SPLINE
SPL {X  -159.452, Y  +378.767, Z    +0.000, E1   +11.887, E3 +156362.622}
SPL {X  -159.840, Y  +384.856, Z    +0.000, E1    +7.126, E3 +156381.593}
SPL {X  -159.991, Y  +390.336, Z    +0.000, E1    +2.803, E3 +156395.416}
SPL {X  -160.000, Y  +403.532, Z    +0.000, E1    -6.523, E3 +156413.137}
SPL {X  -160.000, Y  +409.023, Z    +0.000, E1   -10.003, E3 +156423.910}
SPL {X  -160.000, Y  +418.032, Z    +0.000, E1   -14.569, E3 +156448.770}
SPL {X  -160.000, Y  +420.561, Z    +0.000, E1   -14.816, E3 +156466.250}
SPL {X  -160.000, Y  +422.801, Z    +0.000, E1   -14.823, E3 +156484.198}
SPL {X  -160.000, Y  +425.518, Z    +0.000, E1   -14.845, E3 +156505.973}
SPL {X  -160.000, Y  +428.688, Z    +0.000, E1   -14.854, E3 +156531.381}
SPL {X  -160.000, Y  +431.971, Z    +0.000, E1   -14.849, E3 +156557.850}
SPL {X  -160.000, Y  +435.345, Z    +0.000, E1   -14.857, E3 +156584.900}
SPL {X  -160.000, Y  +438.732, Z    +0.000, E1   -14.858, E3 +156612.048}
SPL {X  -160.000, Y  +441.925, Z    +0.000, E1   -14.848, E3 +156637.718}
SPL {X  -160.000, Y  +444.299, Z    +0.000, E1   -14.809, E3 +156656.903}
SPL {X  -160.000, Y  +446.229, Z    +0.000, E1   -14.820, E3 +156672.322}
SPL {X  -160.000, Y  +448.987, Z    +0.000, E1   -14.868, E3 +156694.259}
SPL {X  -160.000, Y  +452.351, Z    +0.000, E1   -14.871, E3 +156721.235}
SPL {X  -160.000, Y  +455.709, Z    +0.000, E1   -14.880, E3 +156748.049}
SPL {X  -160.000, Y  +458.189, Z    +0.000, E1   -14.832, E3 +156768.051}
SPL {X  -160.000, Y  +459.885, Z    +0.000, E1   -14.825, E3 +156781.721}
SPL {X  -160.000, Y  +462.438, Z    +0.000, E1   -14.868, E3 +156802.131}
SPL {X  -160.000, Y  +465.575, Z    +0.000, E1   -14.849, E3 +156827.439}
SPL {X  -160.000, Y  +468.581, Z    +0.000, E1   -14.841, E3 +156851.672}
SPL {X  -160.000, Y  +471.795, Z    +0.000, E1   -14.854, E3 +156877.459}
SPL {X  -160.000, Y  +475.138, Z    +0.000, E1   -14.853, E3 +156904.310}
SPL {X  -160.000, Y  +477.981, Z    +0.000, E1   -14.823, E3 +156927.230}
SPL {X  -160.000, Y  +480.658, Z    +0.000, E1   -14.835, E3 +156948.706}
SPL {X  -160.000, Y  +483.534, Z    +0.000, E1   -14.838, E3 +156971.801}
SPL {X  -160.000, Y  +486.226, Z    +0.000, E1   -14.823, E3 +156993.466}
SPL {X  -160.000, Y  +488.751, Z    +0.000, E1   -14.827, E3 +157013.738}
SPL {X  -160.000, Y  +491.612, Z    +0.000, E1   -14.844, E3 +157036.661}
SPL {X  -160.000, Y  +494.417, Z    +0.000, E1   -14.827, E3 +157059.252}
SPL {X  -160.000, Y  +496.961, Z    +0.000, E1   -14.824, E3 +157079.696}
SPL {X  -160.000, Y  +499.610, Z    +0.000, E1   -14.830, E3 +157100.968}
SPL {X  -160.000, Y  +502.268, Z    +0.000, E1   -14.832, E3 +157122.238}
SPL {X  -160.000, Y  +505.041, Z    +0.000, E1   -14.849, E3 +157144.400}
SPL {X  -160.000, Y  +507.743, Z    +0.000, E1   -14.842, E3 +157166.024}
SPL {X  -160.000, Y  +510.437, Z    +0.000, E1   -14.860, E3 +157187.538}
SPL {X  -160.000, Y  +513.179, Z    +0.000, E1   -14.849, E3 +157209.585}
SPL {X  -160.000, Y  +515.613, Z    +0.000, E1   -14.829, E3 +157229.256}
SPL {X  -160.000, Y  +518.188, Z    +0.000, E1   -14.845, E3 +157249.885}
SPL {X  -160.000, Y  +520.790, Z    +0.000, E1   -14.839, E3 +157270.714}
SPL {X  -160.000, Y  +523.469, Z    +0.000, E1   -14.855, E3 +157292.162}
SPL {X  -160.000, Y  +526.403, Z    +0.000, E1   -14.858, E3 +157315.698}
SPL {X  -160.000, Y  +529.266, Z    +0.000, E1   -14.848, E3 +157338.706}
SPL {X  -160.000, Y  +531.688, Z    +0.000, E1   -14.826, E3 +157358.255}
SPL {X  -160.000, Y  +534.214, Z    +0.000, E1   -14.841, E3 +157378.518}
SPL {X  -160.000, Y  +537.002, Z    +0.000, E1   -14.839, E3 +157400.937}
SPL {X  -160.000, Y  +539.729, Z    +0.000, E1   -14.840, E3 +157422.748}
SPL {X  -160.000, Y  +542.408, Z    +0.000, E1   -14.839, E3 +157444.301}
SPL {X  -160.000, Y  +545.014, Z    +0.000, E1   -14.831, E3 +157465.246}
SPL {X  -160.000, Y  +547.659, Z    +0.000, E1   -14.839, E3 +157486.461}
SPL {X  -160.000, Y  +550.215, Z    +0.000, E1   -14.827, E3 +157507.026}
SPL {X  -160.000, Y  +552.762, Z    +0.000, E1   -14.836, E3 +157527.444}
SPL {X  -160.000, Y  +555.331, Z    +0.000, E1   -14.837, E3 +157547.985}
SPL {X  -160.000, Y  +558.235, Z    +0.000, E1   -14.869, E3 +157571.149}
SPL {X  -160.000, Y  +561.088, Z    +0.000, E1   -14.848, E3 +157594.067}
SPL {X  -160.000, Y  +563.693, Z    +0.000, E1   -14.852, E3 +157614.928}
SPL {X  -160.000, Y  +566.560, Z    +0.000, E1   -14.865, E3 +157637.905}
SPL {X  -160.000, Y  +569.305, Z    +0.000, E1   -14.848, E3 +157659.934}
SPL {X  -160.000, Y  +571.769, Z    +0.000, E1   -14.852, E3 +157679.680}
SPL {X  -160.000, Y  +574.366, Z    +0.000, E1   -14.855, E3 +157700.467}
SPL {X  -160.000, Y  +577.037, Z    +0.000, E1   -14.859, E3 +157721.866}
SPL {X  -160.000, Y  +579.855, Z    +0.000, E1   -14.869, E3 +157744.393}
SPL {X  -160.000, Y  +582.456, Z    +0.000, E1   -14.854, E3 +157765.253}
SPL {X  -160.000, Y  +585.083, Z    +0.000, E1   -14.866, E3 +157786.303}
SPL {X  -160.000, Y  +587.675, Z    +0.000, E1   -14.853, E3 +157807.094}
SPL {X  -160.000, Y  +590.216, Z    +0.000, E1   -14.864, E3 +157827.413}
SPL {X  -160.000, Y  +592.848, Z    +0.000, E1   -14.865, E3 +157848.464}
SPL {X  -160.000, Y  +595.342, Z    +0.000, E1   -14.848, E3 +157868.642}
SPL {X  -160.000, Y  +597.995, Z    +0.000, E1   -14.848, E3 +157889.982}
SPL {X  -160.000, Y  +600.731, Z    +0.000, E1   -14.846, E3 +157911.933}
SPL {X  -160.000, Y  +603.404, Z    +0.000, E1   -14.846, E3 +157933.369}
SPL {X  -160.000, Y  +605.923, Z    +0.000, E1   -14.838, E3 +157953.610}
SPL {X  -160.000, Y  +608.492, Z    +0.000, E1   -14.846, E3 +157974.214}
SPL {X  -160.000, Y  +611.345, Z    +0.000, E1   -14.856, E3 +157997.072}
SPL {X  -160.000, Y  +614.087, Z    +0.000, E1   -14.839, E3 +158019.131}
SPL {X  -160.000, Y  +616.566, Z    +0.000, E1   -14.839, E3 +158039.025}
SPL {X  -160.000, Y  +619.350, Z    +0.000, E1   -14.855, E3 +158061.313}
SPL {X  -160.000, Y  +622.198, Z    +0.000, E1   -14.846, E3 +158084.197}
SPL {X  -160.000, Y  +624.642, Z    +0.000, E1   -14.829, E3 +158103.870}
SPL {X  -160.000, Y  +627.119, Z    +0.000, E1   -14.843, E3 +158123.710}
SPL {X  -160.000, Y  +629.682, Z    +0.000, E1   -14.838, E3 +158144.279}
SPL {X  -160.000, Y  +632.223, Z    +0.000, E1   -14.841, E3 +158164.670}
SPL {X  -160.000, Y  +634.941, Z    +0.000, E1   -14.846, E3 +158186.468}
SPL {X  -160.000, Y  +637.723, Z    +0.000, E1   -14.844, E3 +158208.812}
SPL {X  -160.000, Y  +640.315, Z    +0.000, E1   -14.836, E3 +158229.610}
SPL {X  -160.000, Y  +643.085, Z    +0.000, E1   -14.865, E3 +158251.661}
SPL {X  -160.000, Y  +645.845, Z    +0.000, E1   -14.848, E3 +158273.849}
SPL {X  -160.000, Y  +648.229, Z    +0.000, E1   -14.834, E3 +158293.059}
SPL {X  -160.000, Y  +650.656, Z    +0.000, E1   -14.835, E3 +158312.615}
SPL {X  -160.000, Y  +653.134, Z    +0.000, E1   -14.827, E3 +158332.542}
SPL {X  -160.000, Y  +655.670, Z    +0.000, E1   -14.841, E3 +158352.836}
SPL {X  -160.000, Y  +658.349, Z    +0.000, E1   -14.842, E3 +158374.312}
SPL {X  -160.000, Y  +660.936, Z    +0.000, E1   -14.838, E3 +158395.064}
SPL {X  -160.000, Y  +663.567, Z    +0.000, E1   -14.845, E3 +158416.194}
SPL {X  -160.000, Y  +666.216, Z    +0.000, E1   -14.832, E3 +158437.511}
SPL {X  -159.997, Y  +668.731, Z    +0.000, E1   -14.834, E3 +158457.703}
SPL {X  -159.962, Y  +671.176, Z    +0.000, E1   -14.822, E3 +158477.414}
SPL {X  -159.895, Y  +673.507, Z    +0.000, E1   -14.821, E3 +158496.145}
SPL {X  -159.785, Y  +675.985, Z    +0.000, E1   -14.818, E3 +158516.147}
SPL {X  -159.627, Y  +678.622, Z    +0.000, E1   -14.804, E3 +158537.500}
SPL {X  -159.438, Y  +681.094, Z    +0.000, E1   -14.770, E3 +158557.671}
SPL {X  -159.262, Y  +683.054, Z    +0.000, E1   -14.719, E3 +158573.899}
ENDSPLINE

SPLINE
SPL {X  -159.661, Y  +678.114, Z    +0.000, E1    -9.575, E3 +158603.491}
SPL {X  -159.942, Y  +672.020, Z    +0.000, E1    -4.692, E3 +158622.118}
SPL {X  -160.000, Y  +664.971, Z    +0.000, E1    +0.516, E3 +158641.668}
SPL {X  -160.000, Y  +660.032, Z    +0.000, E1    +3.995, E3 +158653.611}
SPL {X  -160.000, Y  +652.280, Z    +0.000, E1    +8.913, E3 +158672.126}
SPL {X  -160.000, Y  +644.147, Z    +0.000, E1   +13.158, E3 +158695.677}
SPL {X  -160.000, Y  +641.594, Z    +0.000, E1   +13.488, E3 +158714.118}
SPL {X  -160.000, Y  +639.799, Z    +0.000, E1   +13.486, E3 +158730.028}
SPL {X  -160.000, Y  +637.896, Z    +0.000, E1   +13.493, E3 +158746.843}
SPL {X  -160.000, Y  +635.832, Z    +0.000, E1   +13.499, E3 +158765.102}
SPL {X  -160.000, Y  +633.839, Z    +0.000, E1   +13.489, E3 +158782.790}
SPL {X  -160.000, Y  +631.625, Z    +0.000, E1   +13.508, E3 +158802.331}
SPL {X  -160.000, Y  +629.417, Z    +0.000, E1   +13.491, E3 +158821.943}
SPL {X  -160.000, Y  +627.180, Z    +0.000, E1   +13.508, E3 +158841.697}
SPL {X  -160.000, Y  +624.970, Z    +0.000, E1   +13.490, E3 +158861.347}
SPL {X  -160.000, Y  +623.020, Z    +0.000, E1   +13.491, E3 +158878.576}
SPL {X  -160.000, Y  +620.888, Z    +0.000, E1   +13.501, E3 +158897.439}
SPL {X  -160.000, Y  +618.790, Z    +0.000, E1   +13.488, E3 +158916.061}
SPL {X  -160.000, Y  +616.631, Z    +0.000, E1   +13.504, E3 +158935.115}
SPL {X  -160.000, Y  +614.230, Z    +0.000, E1   +13.510, E3 +158956.311}
SPL {X  -160.000, Y  +612.132, Z    +0.000, E1   +13.485, E3 +158975.027}
SPL {X  -160.000, Y  +610.405, Z    +0.000, E1   +13.477, E3 +158990.400}
SPL {X  -160.000, Y  +608.437, Z    +0.000, E1   +13.502, E3 +159007.656}
SPL {X  -160.000, Y  +606.281, Z    +0.000, E1   +13.502, E3 +159026.673}
SPL {X  -160.000, Y  +604.124, Z    +0.000, E1   +13.513, E3 +159045.729}
SPL {X  -160.000, Y  +601.878, Z    +0.000, E1   +13.505, E3 +159065.626}
SPL {X  -160.000, Y  +599.648, Z    +0.000, E1   +13.506, E3 +159085.403}
SPL {X  -160.000, Y  +597.673, Z    +0.000, E1   +13.479, E3 +159103.076}
SPL {X  -160.000, Y  +595.601, Z    +0.000, E1   +13.499, E3 +159121.359}
SPL {X  -160.000, Y  +593.187, Z    +0.000, E1   +13.500, E3 +159142.739}
SPL {X  -160.000, Y  +591.079, Z    +0.000, E1   +13.483, E3 +159161.466}
SPL {X  -160.000, Y  +589.151, Z    +0.000, E1   +13.489, E3 +159178.517}
SPL {X  -160.000, Y  +586.908, Z    +0.000, E1   +13.501, E3 +159198.362}
SPL {X  -160.000, Y  +584.660, Z    +0.000, E1   +13.490, E3 +159218.304}
SPL {X  -160.000, Y  +582.409, Z    +0.000, E1   +13.499, E3 +159238.222}
SPL {X  -160.000, Y  +580.150, Z    +0.000, E1   +13.490, E3 +159258.268}
SPL {X  -160.000, Y  +577.953, Z    +0.000, E1   +13.493, E3 +159277.727}
SPL {X  -160.000, Y  +575.630, Z    +0.000, E1   +13.502, E3 +159298.211}
SPL {X  -160.000, Y  +573.418, Z    +0.000, E1   +13.502, E3 +159317.719}
SPL {X  -160.000, Y  +571.226, Z    +0.000, E1   +13.520, E3 +159336.927}
SPL {X  -160.000, Y  +569.166, Z    +0.000, E1   +13.512, E3 +159355.118}
SPL {X  -160.000, Y  +567.275, Z    +0.000, E1   +13.517, E3 +159371.785}
SPL {X  -160.000, Y  +565.259, Z    +0.000, E1   +13.523, E3 +159389.574}
SPL {X  -160.000, Y  +563.305, Z    +0.000, E1   +13.512, E3 +159406.913}
SPL {X  -160.000, Y  +561.240, Z    +0.000, E1   +13.521, E3 +159425.174}
SPL {X  -160.000, Y  +558.881, Z    +0.000, E1   +13.524, E3 +159446.016}
SPL {X  -160.000, Y  +556.697, Z    +0.000, E1   +13.510, E3 +159465.402}
SPL {X  -160.000, Y  +554.624, Z    +0.000, E1   +13.512, E3 +159483.733}
SPL {X  -160.000, Y  +552.465, Z    +0.000, E1   +13.514, E3 +159502.818}
SPL {X  -160.000, Y  +550.315, Z    +0.000, E1   +13.514, E3 +159521.811}
SPL {X  -160.000, Y  +548.056, Z    +0.000, E1   +13.519, E3 +159541.812}
SPL {X  -160.000, Y  +545.826, Z    +0.000, E1   +13.501, E3 +159561.690}
SPL {X  -160.000, Y  +543.677, Z    +0.000, E1   +13.502, E3 +159580.748}
SPL {X  -160.000, Y  +541.664, Z    +0.000, E1   +13.489, E3 +159598.633}
SPL {X  -160.000, Y  +539.659, Z    +0.000, E1   +13.494, E3 +159616.393}
SPL {X  -160.000, Y  +537.370, Z    +0.000, E1   +13.501, E3 +159636.632}
SPL {X  -160.000, Y  +535.056, Z    +0.000, E1   +13.506, E3 +159657.028}
SPL {X  -160.000, Y  +532.975, Z    +0.000, E1   +13.494, E3 +159675.515}
SPL {X  -160.000, Y  +530.925, Z    +0.000, E1   +13.499, E3 +159693.676}
SPL {X  -160.000, Y  +528.768, Z    +0.000, E1   +13.498, E3 +159712.778}
SPL {X  -160.000, Y  +526.547, Z    +0.000, E1   +13.499, E3 +159732.446}
SPL {X  -160.000, Y  +523.964, Z    +0.000, E1   +13.742, E3 +159751.951}
SPL {X  -160.000, Y  +513.971, Z    +0.000, E1   +18.644, E3 +159770.863}
SPL {X  -160.000, Y  +513.562, Z    +0.000, E1   +16.972, E3 +159790.740}
SPL {X  -160.000, Y  +513.358, Z    +0.000, E1   +15.267, E3 +159811.012}
SPL {X  -160.000, Y  +512.244, Z    +0.000, E1   +14.473, E3 +159829.468}
SPL {X  -160.000, Y  +509.675, Z    +0.000, E1   +14.481, E3 +159850.611}
SPL {X  -160.000, Y  +507.162, Z    +0.000, E1   +14.470, E3 +159871.351}
SPL {X  -160.000, Y  +504.735, Z    +0.000, E1   +14.473, E3 +159891.323}
SPL {X  -160.000, Y  +502.261, Z    +0.000, E1   +14.476, E3 +159911.659}
SPL {X  -160.000, Y  +499.798, Z    +0.000, E1   +14.482, E3 +159931.861}
SPL {X  -160.000, Y  +497.435, Z    +0.000, E1   +14.476, E3 +159951.338}
SPL {X  -160.000, Y  +495.089, Z    +0.000, E1   +14.475, E3 +159970.705}
SPL {X  -160.000, Y  +492.764, Z    +0.000, E1   +14.469, E3 +159989.876}
SPL {X  -160.000, Y  +490.292, Z    +0.000, E1   +14.476, E3 +160010.277}
SPL {X  -160.000, Y  +487.641, Z    +0.000, E1   +14.470, E3 +160032.173}
SPL {X  -160.000, Y  +485.054, Z    +0.000, E1   +14.460, E3 +160053.616}
SPL {X  -160.000, Y  +482.421, Z    +0.000, E1   +14.461, E3 +160075.334}
SPL {X  -160.000, Y  +480.000, Z    +0.000, E1   +14.451, E3 +160095.298}
SPL {X  -160.000, Y  +477.551, Z    +0.000, E1   +14.466, E3 +160115.427}
SPL {X  -160.000, Y  +475.253, Z    +0.000, E1   +14.450, E3 +160134.401}
SPL {X  -160.000, Y  +473.070, Z    +0.000, E1   +14.454, E3 +160152.422}
SPL {X  -160.000, Y  +470.603, Z    +0.000, E1   +14.464, E3 +160172.722}
SPL {X  -160.000, Y  +468.243, Z    +0.000, E1   +14.458, E3 +160192.121}
SPL {X  -160.000, Y  +465.791, Z    +0.000, E1   +14.475, E3 +160212.265}
SPL {X  -160.000, Y  +463.103, Z    +0.000, E1   +14.474, E3 +160234.414}
SPL {X  -160.000, Y  +460.743, Z    +0.000, E1   +14.465, E3 +160253.822}
SPL {X  -160.000, Y  +458.292, Z    +0.000, E1   +14.492, E3 +160273.822}
SPL {X  -160.000, Y  +455.874, Z    +0.000, E1   +14.484, E3 +160293.679}
SPL {X  -160.000, Y  +453.555, Z    +0.000, E1   +14.488, E3 +160312.759}
SPL {X  -160.000, Y  +451.093, Z    +0.000, E1   +14.485, E3 +160333.071}
SPL {X  -160.000, Y  +448.700, Z    +0.000, E1   +14.483, E3 +160352.760}
SPL {X  -160.000, Y  +446.277, Z    +0.000, E1   +14.485, E3 +160372.684}
SPL {X  -160.000, Y  +443.879, Z    +0.000, E1   +14.485, E3 +160392.422}
SPL {X  -160.000, Y  +441.447, Z    +0.000, E1   +14.485, E3 +160412.429}
SPL {X  -160.000, Y  +439.006, Z    +0.000, E1   +14.488, E3 +160432.512}
SPL {X  -160.000, Y  +436.311, Z    +0.000, E1   +14.498, E3 +160454.671}
SPL {X  -160.000, Y  +433.559, Z    +0.000, E1   +14.491, E3 +160477.341}
SPL {X  -160.000, Y  +431.162, Z    +0.000, E1   +14.479, E3 +160497.092}
SPL {X  -160.000, Y  +429.152, Z    +0.000, E1   +14.469, E3 +160513.673}
SPL {X  -160.000, Y  +426.863, Z    +0.000, E1   +14.490, E3 +160532.452}
SPL {X  -160.000, Y  +424.653, Z    +0.000, E1   +14.467, E3 +160550.712}
SPL {X  -160.000, Y  +422.337, Z    +0.000, E1   +14.492, E3 +160569.696}
SPL {X  -160.000, Y  +419.639, Z    +0.000, E1   +14.504, E3 +160591.736}
SPL {X  -160.000, Y  +417.127, Z    +0.000, E1   +14.501, E3 +160612.327}
SPL {X  -160.000, Y  +414.849, Z    +0.000, E1   +14.496, E3 +160631.061}
SPL {X  -160.000, Y  +412.396, Z    +0.000, E1   +14.505, E3 +160651.250}
SPL {X  -160.000, Y  +409.815, Z    +0.000, E1   +14.498, E3 +160672.504}
SPL {X  -160.000, Y  +407.614, Z    +0.000, E1   +14.484, E3 +160690.629}
SPL {X  -160.000, Y  +405.406, Z    +0.000, E1   +14.501, E3 +160708.692}
SPL {X  -160.000, Y  +402.958, Z    +0.000, E1   +14.500, E3 +160728.862}
SPL {X  -160.000, Y  +400.690, Z    +0.000, E1   +14.484, E3 +160747.574}
SPL {X  -160.000, Y  +398.391, Z    +0.000, E1   +14.502, E3 +160766.400}
SPL {X  -160.000, Y  +395.999, Z    +0.000, E1   +14.484, E3 +160786.190}
SPL {X  -160.000, Y  +393.685, Z    +0.000, E1   +14.486, E3 +160805.262}
SPL {X  -159.999, Y  +391.313, Z    +0.000, E1   +14.479, E3 +160824.844}
SPL {X  -159.970, Y  +388.900, Z    +0.000, E1   +14.480, E3 +160844.729}
SPL {X  -159.903, Y  +386.417, Z    +0.000, E1   +14.475, E3 +160865.234}
SPL {X  -159.796, Y  +383.921, Z    +0.000, E1   +14.466, E3 +160885.889}
SPL {X  -159.651, Y  +381.443, Z    +0.000, E1   +14.453, E3 +160906.437}
SPL {X  -159.474, Y  +379.042, Z    +0.000, E1   +14.434, E3 +160926.401}
SPL {X  -159.316, Y  +377.219, Z    +0.000, E1   +14.400, E3 +160941.629}
ENDSPLINE

SPLINE
SPL {X  -159.452, Y  +378.767, Z    +0.000, E1   +11.887, E3 +160962.619}
SPL {X  -159.840, Y  +384.856, Z    +0.000, E1    +7.126, E3 +160981.590}
SPL {X  -159.991, Y  +390.336, Z    +0.000, E1    +2.803, E3 +160995.413}
SPL {X  -160.000, Y  +403.532, Z    +0.000, E1    -6.523, E3 +161013.134}
SPL {X  -160.000, Y  +409.023, Z    +0.000, E1   -10.003, E3 +161023.907}
SPL {X  -160.000, Y  +418.032, Z    +0.000, E1   -14.569, E3 +161048.766}
SPL {X  -160.000, Y  +420.561, Z    +0.000, E1   -14.816, E3 +161066.246}
SPL {X  -160.000, Y  +422.801, Z    +0.000, E1   -14.823, E3 +161084.195}
SPL {X  -160.000, Y  +425.518, Z    +0.000, E1   -14.845, E3 +161105.970}
SPL {X  -160.000, Y  +428.688, Z    +0.000, E1   -14.854, E3 +161131.378}
SPL {X  -160.000, Y  +431.971, Z    +0.000, E1   -14.849, E3 +161157.846}
SPL {X  -160.000, Y  +435.345, Z    +0.000, E1   -14.857, E3 +161184.897}
SPL {X  -160.000, Y  +438.732, Z    +0.000, E1   -14.858, E3 +161212.045}
SPL {X  -160.000, Y  +441.925, Z    +0.000, E1   -14.848, E3 +161237.715}
SPL {X  -160.000, Y  +444.299, Z    +0.000, E1   -14.809, E3 +161256.900}
SPL {X  -160.000, Y  +446.229, Z    +0.000, E1   -14.820, E3 +161272.319}
SPL {X  -160.000, Y  +448.987, Z    +0.000, E1   -14.868, E3 +161294.256}
SPL {X  -160.000, Y  +452.351, Z    +0.000, E1   -14.871, E3 +161321.232}
SPL {X  -160.000, Y  +455.709, Z    +0.000, E1   -14.880, E3 +161348.046}
SPL {X  -160.000, Y  +458.189, Z    +0.000, E1   -14.832, E3 +161368.047}
SPL {X  -160.000, Y  +459.885, Z    +0.000, E1   -14.825, E3 +161381.718}
SPL {X  -160.000, Y  +462.438, Z    +0.000, E1   -14.868, E3 +161402.128}
SPL {X  -160.000, Y  +465.575, Z    +0.000, E1   -14.849, E3 +161427.436}
SPL {X  -160.000, Y  +468.581, Z    +0.000, E1   -14.841, E3 +161451.669}
SPL {X  -160.000, Y  +471.795, Z    +0.000, E1   -14.854, E3 +161477.456}
SPL {X  -160.000, Y  +475.138, Z    +0.000, E1   -14.853, E3 +161504.306}
SPL {X  -160.000, Y  +477.981, Z    +0.000, E1   -14.823, E3 +161527.227}
SPL {X  -160.000, Y  +480.658, Z    +0.000, E1   -14.835, E3 +161548.703}
SPL {X  -160.000, Y  +483.534, Z    +0.000, E1   -14.838, E3 +161571.798}
SPL {X  -160.000, Y  +486.226, Z    +0.000, E1   -14.823, E3 +161593.463}
SPL {X  -160.000, Y  +488.751, Z    +0.000, E1   -14.827, E3 +161613.735}
SPL {X  -160.000, Y  +491.612, Z    +0.000, E1   -14.844, E3 +161636.658}
SPL {X  -160.000, Y  +494.417, Z    +0.000, E1   -14.827, E3 +161659.249}
SPL {X  -160.000, Y  +496.961, Z    +0.000, E1   -14.824, E3 +161679.692}
SPL {X  -160.000, Y  +499.610, Z    +0.000, E1   -14.830, E3 +161700.965}
SPL {X  -160.000, Y  +502.268, Z    +0.000, E1   -14.832, E3 +161722.234}
SPL {X  -160.000, Y  +505.041, Z    +0.000, E1   -14.849, E3 +161744.397}
SPL {X  -160.000, Y  +507.743, Z    +0.000, E1   -14.842, E3 +161766.021}
SPL {X  -160.000, Y  +510.437, Z    +0.000, E1   -14.860, E3 +161787.535}
SPL {X  -160.000, Y  +513.179, Z    +0.000, E1   -14.849, E3 +161809.582}
SPL {X  -160.000, Y  +515.613, Z    +0.000, E1   -14.829, E3 +161829.252}
SPL {X  -160.000, Y  +518.188, Z    +0.000, E1   -14.845, E3 +161849.882}
SPL {X  -160.000, Y  +520.790, Z    +0.000, E1   -14.839, E3 +161870.711}
SPL {X  -160.000, Y  +523.469, Z    +0.000, E1   -14.855, E3 +161892.159}
SPL {X  -160.000, Y  +526.403, Z    +0.000, E1   -14.858, E3 +161915.695}
SPL {X  -160.000, Y  +529.266, Z    +0.000, E1   -14.848, E3 +161938.702}
SPL {X  -160.000, Y  +531.688, Z    +0.000, E1   -14.826, E3 +161958.252}
SPL {X  -160.000, Y  +534.214, Z    +0.000, E1   -14.841, E3 +161978.515}
SPL {X  -160.000, Y  +537.002, Z    +0.000, E1   -14.839, E3 +162000.933}
SPL {X  -160.000, Y  +539.729, Z    +0.000, E1   -14.840, E3 +162022.745}
SPL {X  -160.000, Y  +542.408, Z    +0.000, E1   -14.839, E3 +162044.298}
SPL {X  -160.000, Y  +545.014, Z    +0.000, E1   -14.831, E3 +162065.243}
SPL {X  -160.000, Y  +547.659, Z    +0.000, E1   -14.839, E3 +162086.458}
SPL {X  -160.000, Y  +550.215, Z    +0.000, E1   -14.827, E3 +162107.023}
SPL {X  -160.000, Y  +552.762, Z    +0.000, E1   -14.836, E3 +162127.441}
SPL {X  -160.000, Y  +555.331, Z    +0.000, E1   -14.837, E3 +162147.982}
SPL {X  -160.000, Y  +558.235, Z    +0.000, E1   -14.869, E3 +162171.145}
SPL {X  -160.000, Y  +561.088, Z    +0.000, E1   -14.848, E3 +162194.064}
SPL {X  -160.000, Y  +563.693, Z    +0.000, E1   -14.852, E3 +162214.924}
SPL {X  -160.000, Y  +566.560, Z    +0.000, E1   -14.865, E3 +162237.902}
SPL {X  -160.000, Y  +569.305, Z    +0.000, E1   -14.848, E3 +162259.931}
SPL {X  -160.000, Y  +571.769, Z    +0.000, E1   -14.852, E3 +162279.676}
SPL {X  -160.000, Y  +574.366, Z    +0.000, E1   -14.855, E3 +162300.463}
SPL {X  -160.000, Y  +577.037, Z    +0.000, E1   -14.859, E3 +162321.863}
SPL {X  -160.000, Y  +579.855, Z    +0.000, E1   -14.869, E3 +162344.390}
SPL {X  -160.000, Y  +582.456, Z    +0.000, E1   -14.854, E3 +162365.250}
SPL {X  -160.000, Y  +585.083, Z    +0.000, E1   -14.866, E3 +162386.300}
SPL {X  -160.000, Y  +587.675, Z    +0.000, E1   -14.853, E3 +162407.091}
SPL {X  -160.000, Y  +590.216, Z    +0.000, E1   -14.864, E3 +162427.410}
SPL {X  -160.000, Y  +592.848, Z    +0.000, E1   -14.865, E3 +162448.461}
SPL {X  -160.000, Y  +595.342, Z    +0.000, E1   -14.848, E3 +162468.639}
SPL {X  -160.000, Y  +597.995, Z    +0.000, E1   -14.848, E3 +162489.979}
SPL {X  -160.000, Y  +600.731, Z    +0.000, E1   -14.846, E3 +162511.930}
SPL {X  -160.000, Y  +603.404, Z    +0.000, E1   -14.846, E3 +162533.366}
SPL {X  -160.000, Y  +605.923, Z    +0.000, E1   -14.838, E3 +162553.607}
SPL {X  -160.000, Y  +608.492, Z    +0.000, E1   -14.846, E3 +162574.210}
SPL {X  -160.000, Y  +611.345, Z    +0.000, E1   -14.856, E3 +162597.069}
SPL {X  -160.000, Y  +614.087, Z    +0.000, E1   -14.839, E3 +162619.128}
SPL {X  -160.000, Y  +616.566, Z    +0.000, E1   -14.839, E3 +162639.022}
SPL {X  -160.000, Y  +619.350, Z    +0.000, E1   -14.855, E3 +162661.310}
SPL {X  -160.000, Y  +622.198, Z    +0.000, E1   -14.846, E3 +162684.194}
SPL {X  -160.000, Y  +624.642, Z    +0.000, E1   -14.829, E3 +162703.867}
SPL {X  -160.000, Y  +627.119, Z    +0.000, E1   -14.843, E3 +162723.707}
SPL {X  -160.000, Y  +629.682, Z    +0.000, E1   -14.838, E3 +162744.276}
SPL {X  -160.000, Y  +632.223, Z    +0.000, E1   -14.841, E3 +162764.667}
SPL {X  -160.000, Y  +634.941, Z    +0.000, E1   -14.846, E3 +162786.465}
SPL {X  -160.000, Y  +637.723, Z    +0.000, E1   -14.844, E3 +162808.809}
SPL {X  -160.000, Y  +640.315, Z    +0.000, E1   -14.836, E3 +162829.606}
SPL {X  -160.000, Y  +643.085, Z    +0.000, E1   -14.865, E3 +162851.658}
SPL {X  -160.000, Y  +645.845, Z    +0.000, E1   -14.848, E3 +162873.846}
SPL {X  -160.000, Y  +648.229, Z    +0.000, E1   -14.834, E3 +162893.056}
SPL {X  -160.000, Y  +650.656, Z    +0.000, E1   -14.835, E3 +162912.612}
SPL {X  -160.000, Y  +653.134, Z    +0.000, E1   -14.827, E3 +162932.539}
SPL {X  -160.000, Y  +655.670, Z    +0.000, E1   -14.841, E3 +162952.833}
SPL {X  -160.000, Y  +658.349, Z    +0.000, E1   -14.842, E3 +162974.309}
SPL {X  -160.000, Y  +660.936, Z    +0.000, E1   -14.838, E3 +162995.061}
SPL {X  -160.000, Y  +663.567, Z    +0.000, E1   -14.845, E3 +163016.191}
SPL {X  -160.000, Y  +666.216, Z    +0.000, E1   -14.832, E3 +163037.508}
SPL {X  -159.997, Y  +668.731, Z    +0.000, E1   -14.834, E3 +163057.700}
SPL {X  -159.962, Y  +671.176, Z    +0.000, E1   -14.822, E3 +163077.411}
SPL {X  -159.895, Y  +673.507, Z    +0.000, E1   -14.821, E3 +163096.142}
SPL {X  -159.785, Y  +675.985, Z    +0.000, E1   -14.818, E3 +163116.144}
SPL {X  -159.627, Y  +678.622, Z    +0.000, E1   -14.804, E3 +163137.496}
SPL {X  -159.438, Y  +681.094, Z    +0.000, E1   -14.770, E3 +163157.668}
SPL {X  -159.262, Y  +683.054, Z    +0.000, E1   -14.719, E3 +163173.896}
ENDSPLINE

SPLINE
SPL {X  -159.661, Y  +678.114, Z    +0.000, E1    -9.575, E3 +163203.488}
SPL {X  -159.942, Y  +672.020, Z    +0.000, E1    -4.692, E3 +163222.115}
SPL {X  -160.000, Y  +664.971, Z    +0.000, E1    +0.516, E3 +163241.665}
SPL {X  -160.000, Y  +660.032, Z    +0.000, E1    +3.995, E3 +163253.608}
SPL {X  -160.000, Y  +652.280, Z    +0.000, E1    +8.913, E3 +163272.123}
SPL {X  -160.000, Y  +644.147, Z    +0.000, E1   +13.158, E3 +163295.674}
SPL {X  -160.000, Y  +641.594, Z    +0.000, E1   +13.488, E3 +163314.115}
SPL {X  -160.000, Y  +639.799, Z    +0.000, E1   +13.486, E3 +163330.025}
SPL {X  -160.000, Y  +637.896, Z    +0.000, E1   +13.493, E3 +163346.840}
SPL {X  -160.000, Y  +635.832, Z    +0.000, E1   +13.499, E3 +163365.098}
SPL {X  -160.000, Y  +633.839, Z    +0.000, E1   +13.489, E3 +163382.787}
SPL {X  -160.000, Y  +631.625, Z    +0.000, E1   +13.508, E3 +163402.328}
SPL {X  -160.000, Y  +629.417, Z    +0.000, E1   +13.491, E3 +163421.939}
SPL {X  -160.000, Y  +627.180, Z    +0.000, E1   +13.508, E3 +163441.693}
SPL {X  -160.000, Y  +624.970, Z    +0.000, E1   +13.490, E3 +163461.343}
SPL {X  -160.000, Y  +623.020, Z    +0.000, E1   +13.491, E3 +163478.573}
SPL {X  -160.000, Y  +620.888, Z    +0.000, E1   +13.501, E3 +163497.436}
SPL {X  -160.000, Y  +618.790, Z    +0.000, E1   +13.488, E3 +163516.058}
SPL {X  -160.000, Y  +616.631, Z    +0.000, E1   +13.504, E3 +163535.112}
SPL {X  -160.000, Y  +614.230, Z    +0.000, E1   +13.510, E3 +163556.307}
SPL {X  -160.000, Y  +612.132, Z    +0.000, E1   +13.485, E3 +163575.024}
SPL {X  -160.000, Y  +610.405, Z    +0.000, E1   +13.477, E3 +163590.397}
SPL {X  -160.000, Y  +608.437, Z    +0.000, E1   +13.502, E3 +163607.652}
SPL {X  -160.000, Y  +606.281, Z    +0.000, E1   +13.502, E3 +163626.670}
SPL {X  -160.000, Y  +604.124, Z    +0.000, E1   +13.513, E3 +163645.725}
SPL {X  -160.000, Y  +601.878, Z    +0.000, E1   +13.505, E3 +163665.623}
SPL {X  -160.000, Y  +599.648, Z    +0.000, E1   +13.506, E3 +163685.399}
SPL {X  -160.000, Y  +597.673, Z    +0.000, E1   +13.479, E3 +163703.073}
SPL {X  -160.000, Y  +595.601, Z    +0.000, E1   +13.499, E3 +163721.356}
SPL {X  -160.000, Y  +593.187, Z    +0.000, E1   +13.500, E3 +163742.736}
SPL {X  -160.000, Y  +591.079, Z    +0.000, E1   +13.483, E3 +163761.462}
SPL {X  -160.000, Y  +589.151, Z    +0.000, E1   +13.489, E3 +163778.513}
SPL {X  -160.000, Y  +586.908, Z    +0.000, E1   +13.501, E3 +163798.359}
SPL {X  -160.000, Y  +584.660, Z    +0.000, E1   +13.490, E3 +163818.300}
SPL {X  -160.000, Y  +582.409, Z    +0.000, E1   +13.499, E3 +163838.219}
SPL {X  -160.000, Y  +580.150, Z    +0.000, E1   +13.490, E3 +163858.265}
SPL {X  -160.000, Y  +577.953, Z    +0.000, E1   +13.493, E3 +163877.723}
SPL {X  -160.000, Y  +575.630, Z    +0.000, E1   +13.502, E3 +163898.207}
SPL {X  -160.000, Y  +573.418, Z    +0.000, E1   +13.502, E3 +163917.715}
SPL {X  -160.000, Y  +571.226, Z    +0.000, E1   +13.520, E3 +163936.924}
SPL {X  -160.000, Y  +569.166, Z    +0.000, E1   +13.512, E3 +163955.115}
SPL {X  -160.000, Y  +567.275, Z    +0.000, E1   +13.517, E3 +163971.782}
SPL {X  -160.000, Y  +565.259, Z    +0.000, E1   +13.523, E3 +163989.571}
SPL {X  -160.000, Y  +563.305, Z    +0.000, E1   +13.512, E3 +164006.909}
SPL {X  -160.000, Y  +561.240, Z    +0.000, E1   +13.521, E3 +164025.171}
SPL {X  -160.000, Y  +558.881, Z    +0.000, E1   +13.524, E3 +164046.013}
SPL {X  -160.000, Y  +556.697, Z    +0.000, E1   +13.510, E3 +164065.399}
SPL {X  -160.000, Y  +554.624, Z    +0.000, E1   +13.512, E3 +164083.730}
SPL {X  -160.000, Y  +552.465, Z    +0.000, E1   +13.514, E3 +164102.814}
SPL {X  -160.000, Y  +550.315, Z    +0.000, E1   +13.514, E3 +164121.808}
SPL {X  -160.000, Y  +548.056, Z    +0.000, E1   +13.519, E3 +164141.809}
SPL {X  -160.000, Y  +545.826, Z    +0.000, E1   +13.501, E3 +164161.687}
SPL {X  -160.000, Y  +543.677, Z    +0.000, E1   +13.502, E3 +164180.745}
SPL {X  -160.000, Y  +541.664, Z    +0.000, E1   +13.489, E3 +164198.630}
SPL {X  -160.000, Y  +539.659, Z    +0.000, E1   +13.494, E3 +164216.390}
SPL {X  -160.000, Y  +537.370, Z    +0.000, E1   +13.501, E3 +164236.629}
SPL {X  -160.000, Y  +535.056, Z    +0.000, E1   +13.506, E3 +164257.025}
SPL {X  -160.000, Y  +532.975, Z    +0.000, E1   +13.494, E3 +164275.511}
SPL {X  -160.000, Y  +530.925, Z    +0.000, E1   +13.499, E3 +164293.673}
SPL {X  -160.000, Y  +528.768, Z    +0.000, E1   +13.498, E3 +164312.775}
SPL {X  -160.000, Y  +526.547, Z    +0.000, E1   +13.499, E3 +164332.443}
SPL {X  -160.000, Y  +523.964, Z    +0.000, E1   +13.742, E3 +164351.948}
SPL {X  -160.000, Y  +513.971, Z    +0.000, E1   +18.644, E3 +164370.860}
SPL {X  -160.000, Y  +513.562, Z    +0.000, E1   +16.972, E3 +164390.736}
SPL {X  -160.000, Y  +513.358, Z    +0.000, E1   +15.267, E3 +164411.008}
SPL {X  -160.000, Y  +512.244, Z    +0.000, E1   +14.473, E3 +164429.465}
SPL {X  -160.000, Y  +509.675, Z    +0.000, E1   +14.481, E3 +164450.608}
SPL {X  -160.000, Y  +507.162, Z    +0.000, E1   +14.470, E3 +164471.348}
SPL {X  -160.000, Y  +504.735, Z    +0.000, E1   +14.473, E3 +164491.320}
SPL {X  -160.000, Y  +502.261, Z    +0.000, E1   +14.476, E3 +164511.656}
SPL {X  -160.000, Y  +499.798, Z    +0.000, E1   +14.482, E3 +164531.858}
SPL {X  -160.000, Y  +497.435, Z    +0.000, E1   +14.476, E3 +164551.335}
SPL {X  -160.000, Y  +495.089, Z    +0.000, E1   +14.475, E3 +164570.701}
SPL {X  -160.000, Y  +492.764, Z    +0.000, E1   +14.469, E3 +164589.873}
SPL {X  -160.000, Y  +490.292, Z    +0.000, E1   +14.476, E3 +164610.274}
SPL {X  -160.000, Y  +487.641, Z    +0.000, E1   +14.470, E3 +164632.170}
SPL {X  -160.000, Y  +485.054, Z    +0.000, E1   +14.460, E3 +164653.612}
SPL {X  -160.000, Y  +482.421, Z    +0.000, E1   +14.461, E3 +164675.331}
SPL {X  -160.000, Y  +480.000, Z    +0.000, E1   +14.451, E3 +164695.295}
SPL {X  -160.000, Y  +477.551, Z    +0.000, E1   +14.466, E3 +164715.423}
SPL {X  -160.000, Y  +475.253, Z    +0.000, E1   +14.450, E3 +164734.398}
SPL {X  -160.000, Y  +473.070, Z    +0.000, E1   +14.454, E3 +164752.419}
SPL {X  -160.000, Y  +470.603, Z    +0.000, E1   +14.464, E3 +164772.719}
SPL {X  -160.000, Y  +468.243, Z    +0.000, E1   +14.458, E3 +164792.118}
SPL {X  -160.000, Y  +465.791, Z    +0.000, E1   +14.475, E3 +164812.262}
SPL {X  -160.000, Y  +463.103, Z    +0.000, E1   +14.474, E3 +164834.411}
SPL {X  -160.000, Y  +460.743, Z    +0.000, E1   +14.465, E3 +164853.819}
SPL {X  -160.000, Y  +458.292, Z    +0.000, E1   +14.492, E3 +164873.819}
SPL {X  -160.000, Y  +455.874, Z    +0.000, E1   +14.484, E3 +164893.676}
SPL {X  -160.000, Y  +453.555, Z    +0.000, E1   +14.488, E3 +164912.755}
SPL {X  -160.000, Y  +451.093, Z    +0.000, E1   +14.485, E3 +164933.068}
SPL {X  -160.000, Y  +448.700, Z    +0.000, E1   +14.483, E3 +164952.757}
SPL {X  -160.000, Y  +446.277, Z    +0.000, E1   +14.485, E3 +164972.681}
SPL {X  -160.000, Y  +443.879, Z    +0.000, E1   +14.485, E3 +164992.419}
SPL {X  -160.000, Y  +441.447, Z    +0.000, E1   +14.485, E3 +165012.426}
SPL {X  -160.000, Y  +439.006, Z    +0.000, E1   +14.488, E3 +165032.509}
SPL {X  -160.000, Y  +436.311, Z    +0.000, E1   +14.498, E3 +165054.668}
SPL {X  -160.000, Y  +433.559, Z    +0.000, E1   +14.491, E3 +165077.337}
SPL {X  -160.000, Y  +431.162, Z    +0.000, E1   +14.479, E3 +165097.089}
SPL {X  -160.000, Y  +429.152, Z    +0.000, E1   +14.469, E3 +165113.670}
SPL {X  -160.000, Y  +426.863, Z    +0.000, E1   +14.490, E3 +165132.449}
SPL {X  -160.000, Y  +424.653, Z    +0.000, E1   +14.467, E3 +165150.708}
SPL {X  -160.000, Y  +422.337, Z    +0.000, E1   +14.492, E3 +165169.693}
SPL {X  -160.000, Y  +419.639, Z    +0.000, E1   +14.504, E3 +165191.732}
SPL {X  -160.000, Y  +417.127, Z    +0.000, E1   +14.501, E3 +165212.324}
SPL {X  -160.000, Y  +414.849, Z    +0.000, E1   +14.496, E3 +165231.058}
SPL {X  -160.000, Y  +412.396, Z    +0.000, E1   +14.505, E3 +165251.247}
SPL {X  -160.000, Y  +409.815, Z    +0.000, E1   +14.498, E3 +165272.501}
SPL {X  -160.000, Y  +407.614, Z    +0.000, E1   +14.484, E3 +165290.626}
SPL {X  -160.000, Y  +405.406, Z    +0.000, E1   +14.501, E3 +165308.689}
SPL {X  -160.000, Y  +402.958, Z    +0.000, E1   +14.500, E3 +165328.859}
SPL {X  -160.000, Y  +400.690, Z    +0.000, E1   +14.484, E3 +165347.571}
SPL {X  -160.000, Y  +398.391, Z    +0.000, E1   +14.502, E3 +165366.397}
SPL {X  -160.000, Y  +395.999, Z    +0.000, E1   +14.484, E3 +165386.187}
SPL {X  -160.000, Y  +393.685, Z    +0.000, E1   +14.486, E3 +165405.259}
SPL {X  -159.999, Y  +391.313, Z    +0.000, E1   +14.479, E3 +165424.841}
SPL {X  -159.970, Y  +388.900, Z    +0.000, E1   +14.480, E3 +165444.725}
SPL {X  -159.903, Y  +386.417, Z    +0.000, E1   +14.475, E3 +165465.231}
SPL {X  -159.796, Y  +383.921, Z    +0.000, E1   +14.466, E3 +165485.886}
SPL {X  -159.651, Y  +381.443, Z    +0.000, E1   +14.453, E3 +165506.434}
SPL {X  -159.474, Y  +379.042, Z    +0.000, E1   +14.434, E3 +165526.398}
SPL {X  -159.316, Y  +377.219, Z    +0.000, E1   +14.400, E3 +165541.626}
ENDSPLINE

SPLINE
SPL {X  -159.452, Y  +378.767, Z    +0.000, E1   +11.887, E3 +165562.615}
SPL {X  -159.840, Y  +384.856, Z    +0.000, E1    +7.126, E3 +165581.587}
SPL {X  -159.991, Y  +390.336, Z    +0.000, E1    +2.803, E3 +165595.410}
SPL {X  -160.000, Y  +403.532, Z    +0.000, E1    -6.523, E3 +165613.130}
SPL {X  -160.000, Y  +409.023, Z    +0.000, E1   -10.003, E3 +165623.904}
SPL {X  -160.000, Y  +418.032, Z    +0.000, E1   -14.569, E3 +165648.763}
SPL {X  -160.000, Y  +420.561, Z    +0.000, E1   -14.816, E3 +165666.243}
SPL {X  -160.000, Y  +422.801, Z    +0.000, E1   -14.823, E3 +165684.192}
SPL {X  -160.000, Y  +425.518, Z    +0.000, E1   -14.845, E3 +165705.966}
SPL {X  -160.000, Y  +428.688, Z    +0.000, E1   -14.854, E3 +165731.375}
SPL {X  -160.000, Y  +431.971, Z    +0.000, E1   -14.849, E3 +165757.843}
SPL {X  -160.000, Y  +435.345, Z    +0.000, E1   -14.857, E3 +165784.893}
SPL {X  -160.000, Y  +438.732, Z    +0.000, E1   -14.858, E3 +165812.042}
SPL {X  -160.000, Y  +441.925, Z    +0.000, E1   -14.848, E3 +165837.712}
SPL {X  -160.000, Y  +444.299, Z    +0.000, E1   -14.809, E3 +165856.897}
SPL {X  -160.000, Y  +446.229, Z    +0.000, E1   -14.820, E3 +165872.316}
SPL {X  -160.000, Y  +448.987, Z    +0.000, E1   -14.868, E3 +165894.252}
SPL {X  -160.000, Y  +452.351, Z    +0.000, E1   -14.871, E3 +165921.228}
SPL {X  -160.000, Y  +455.709, Z    +0.000, E1   -14.880, E3 +165948.043}
SPL {X  -160.000, Y  +458.189, Z    +0.000, E1   -14.832, E3 +165968.044}
SPL {X  -160.000, Y  +459.885, Z    +0.000, E1   -14.825, E3 +165981.715}
SPL {X  -160.000, Y  +462.438, Z    +0.000, E1   -14.868, E3 +166002.125}
SPL {X  -160.000, Y  +465.575, Z    +0.000, E1   -14.849, E3 +166027.433}
SPL {X  -160.000, Y  +468.581, Z    +0.000, E1   -14.841, E3 +166051.665}
SPL {X  -160.000, Y  +471.795, Z    +0.000, E1   -14.854, E3 +166077.453}
SPL {X  -160.000, Y  +475.138, Z    +0.000, E1   -14.853, E3 +166104.303}
SPL {X  -160.000, Y  +477.981, Z    +0.000, E1   -14.823, E3 +166127.223}
SPL {X  -160.000, Y  +480.658, Z    +0.000, E1   -14.835, E3 +166148.700}
SPL {X  -160.000, Y  +483.534, Z    +0.000, E1   -14.838, E3 +166171.794}
SPL {X  -160.000, Y  +486.226, Z    +0.000, E1   -14.823, E3 +166193.459}
SPL {X  -160.000, Y  +488.751, Z    +0.000, E1   -14.827, E3 +166213.732}
SPL {X  -160.000, Y  +491.612, Z    +0.000, E1   -14.844, E3 +166236.655}
SPL {X  -160.000, Y  +494.417, Z    +0.000, E1   -14.827, E3 +166259.245}
SPL {X  -160.000, Y  +496.961, Z    +0.000, E1   -14.824, E3 +166279.689}
SPL {X  -160.000, Y  +499.610, Z    +0.000, E1   -14.830, E3 +166300.962}
SPL {X  -160.000, Y  +502.268, Z    +0.000, E1   -14.832, E3 +166322.231}
SPL {X  -160.000, Y  +505.041, Z    +0.000, E1   -14.849, E3 +166344.394}
SPL {X  -160.000, Y  +507.743, Z    +0.000, E1   -14.842, E3 +166366.018}
SPL {X  -160.000, Y  +510.437, Z    +0.000, E1   -14.860, E3 +166387.531}
SPL {X  -160.000, Y  +513.179, Z    +0.000, E1   -14.849, E3 +166409.579}
SPL {X  -160.000, Y  +515.613, Z    +0.000, E1   -14.829, E3 +166429.249}
SPL {X  -160.000, Y  +518.188, Z    +0.000, E1   -14.845, E3 +166449.879}
SPL {X  -160.000, Y  +520.790, Z    +0.000, E1   -14.839, E3 +166470.707}
SPL {X  -160.000, Y  +523.469, Z    +0.000, E1   -14.855, E3 +166492.156}
SPL {X  -160.000, Y  +526.403, Z    +0.000, E1   -14.858, E3 +166515.692}
SPL {X  -160.000, Y  +529.266, Z    +0.000, E1   -14.848, E3 +166538.699}
SPL {X  -160.000, Y  +531.688, Z    +0.000, E1   -14.826, E3 +166558.249}
SPL {X  -160.000, Y  +534.214, Z    +0.000, E1   -14.841, E3 +166578.512}
SPL {X  -160.000, Y  +537.002, Z    +0.000, E1   -14.839, E3 +166600.930}
SPL {X  -160.000, Y  +539.729, Z    +0.000, E1   -14.840, E3 +166622.742}
SPL {X  -160.000, Y  +542.408, Z    +0.000, E1   -14.839, E3 +166644.295}
SPL {X  -160.000, Y  +545.014, Z    +0.000, E1   -14.831, E3 +166665.240}
SPL {X  -160.000, Y  +547.659, Z    +0.000, E1   -14.839, E3 +166686.455}
SPL {X  -160.000, Y  +550.215, Z    +0.000, E1   -14.827, E3 +166707.020}
SPL {X  -160.000, Y  +552.762, Z    +0.000, E1   -14.836, E3 +166727.438}
SPL {X  -160.000, Y  +555.331, Z    +0.000, E1   -14.837, E3 +166747.979}
SPL {X  -160.000, Y  +558.235, Z    +0.000, E1   -14.869, E3 +166771.142}
SPL {X  -160.000, Y  +561.088, Z    +0.000, E1   -14.848, E3 +166794.061}
SPL {X  -160.000, Y  +563.693, Z    +0.000, E1   -14.852, E3 +166814.921}
SPL {X  -160.000, Y  +566.560, Z    +0.000, E1   -14.865, E3 +166837.899}
SPL {X  -160.000, Y  +569.305, Z    +0.000, E1   -14.848, E3 +166859.927}
SPL {X  -160.000, Y  +571.769, Z    +0.000, E1   -14.852, E3 +166879.673}
SPL {X  -160.000, Y  +574.366, Z    +0.000, E1   -14.855, E3 +166900.460}
SPL {X  -160.000, Y  +577.037, Z    +0.000, E1   -14.859, E3 +166921.860}
SPL {X  -160.000, Y  +579.855, Z    +0.000, E1   -14.869, E3 +166944.387}
SPL {X  -160.000, Y  +582.456, Z    +0.000, E1   -14.854, E3 +166965.247}
SPL {X  -160.000, Y  +585.083, Z    +0.000, E1   -14.866, E3 +166986.297}
SPL {X  -160.000, Y  +587.675, Z    +0.000, E1   -14.853, E3 +167007.088}
SPL {X  -160.000, Y  +590.216, Z    +0.000, E1   -14.864, E3 +167027.407}
SPL {X  -160.000, Y  +592.848, Z    +0.000, E1   -14.865, E3 +167048.458}
SPL {X  -160.000, Y  +595.342, Z    +0.000, E1   -14.848, E3 +167068.636}
SPL {X  -160.000, Y  +597.995, Z    +0.000, E1   -14.848, E3 +167089.975}
SPL {X  -160.000, Y  +600.731, Z    +0.000, E1   -14.846, E3 +167111.927}
SPL {X  -160.000, Y  +603.404, Z    +0.000, E1   -14.846, E3 +167133.363}
SPL {X  -160.000, Y  +605.923, Z    +0.000, E1   -14.838, E3 +167153.604}
SPL {X  -160.000, Y  +608.492, Z    +0.000, E1   -14.846, E3 +167174.207}
SPL {X  -160.000, Y  +611.345, Z    +0.000, E1   -14.856, E3 +167197.065}
SPL {X  -160.000, Y  +614.087, Z    +0.000, E1   -14.839, E3 +167219.125}
SPL {X  -160.000, Y  +616.566, Z    +0.000, E1   -14.839, E3 +167239.019}
SPL {X  -160.000, Y  +619.350, Z    +0.000, E1   -14.855, E3 +167261.307}
SPL {X  -160.000, Y  +622.198, Z    +0.000, E1   -14.846, E3 +167284.191}
SPL {X  -160.000, Y  +624.642, Z    +0.000, E1   -14.829, E3 +167303.864}
SPL {X  -160.000, Y  +627.119, Z    +0.000, E1   -14.843, E3 +167323.704}
SPL {X  -160.000, Y  +629.682, Z    +0.000, E1   -14.838, E3 +167344.273}
SPL {X  -160.000, Y  +632.223, Z    +0.000, E1   -14.841, E3 +167364.664}
SPL {X  -160.000, Y  +634.941, Z    +0.000, E1   -14.846, E3 +167386.461}
SPL {X  -160.000, Y  +637.723, Z    +0.000, E1   -14.844, E3 +167408.806}
SPL {X  -160.000, Y  +640.315, Z    +0.000, E1   -14.836, E3 +167429.603}
SPL {X  -160.000, Y  +643.085, Z    +0.000, E1   -14.865, E3 +167451.655}
SPL {X  -160.000, Y  +645.845, Z    +0.000, E1   -14.848, E3 +167473.843}
SPL {X  -160.000, Y  +648.229, Z    +0.000, E1   -14.834, E3 +167493.052}
SPL {X  -160.000, Y  +650.656, Z    +0.000, E1   -14.835, E3 +167512.609}
SPL {X  -160.000, Y  +653.134, Z    +0.000, E1   -14.827, E3 +167532.536}
SPL {X  -160.000, Y  +655.670, Z    +0.000, E1   -14.841, E3 +167552.830}
SPL {X  -160.000, Y  +658.349, Z    +0.000, E1   -14.842, E3 +167574.306}
SPL {X  -160.000, Y  +660.936, Z    +0.000, E1   -14.838, E3 +167595.058}
SPL {X  -160.000, Y  +663.567, Z    +0.000, E1   -14.845, E3 +167616.188}
SPL {X  -160.000, Y  +666.216, Z    +0.000, E1   -14.832, E3 +167637.504}
SPL {X  -159.997, Y  +668.731, Z    +0.000, E1   -14.834, E3 +167657.696}
SPL {X  -159.962, Y  +671.176, Z    +0.000, E1   -14.822, E3 +167677.408}
SPL {X  -159.895, Y  +673.507, Z    +0.000, E1   -14.821, E3 +167696.139}
SPL {X  -159.785, Y  +675.985, Z    +0.000, E1   -14.818, E3 +167716.140}
SPL {X  -159.627, Y  +678.622, Z    +0.000, E1   -14.804, E3 +167737.493}
SPL {X  -159.438, Y  +681.094, Z    +0.000, E1   -14.770, E3 +167757.665}
SPL {X  -159.262, Y  +683.054, Z    +0.000, E1   -14.719, E3 +167773.893}
ENDSPLINE

SPLINE
SPL {X  -159.661, Y  +678.114, Z    +0.000, E1    -9.575, E3 +167803.485}
SPL {X  -159.942, Y  +672.020, Z    +0.000, E1    -4.692, E3 +167822.112}
SPL {X  -160.000, Y  +664.971, Z    +0.000, E1    +0.516, E3 +167841.662}
SPL {X  -160.000, Y  +660.032, Z    +0.000, E1    +3.995, E3 +167853.605}
SPL {X  -160.000, Y  +652.280, Z    +0.000, E1    +8.913, E3 +167872.120}
SPL {X  -160.000, Y  +644.147, Z    +0.000, E1   +13.158, E3 +167895.670}
SPL {X  -160.000, Y  +641.594, Z    +0.000, E1   +13.488, E3 +167914.111}
SPL {X  -160.000, Y  +639.799, Z    +0.000, E1   +13.486, E3 +167930.021}
SPL {X  -160.000, Y  +637.896, Z    +0.000, E1   +13.493, E3 +167946.836}
SPL {X  -160.000, Y  +635.832, Z    +0.000, E1   +13.499, E3 +167965.095}
SPL {X  -160.000, Y  +633.839, Z    +0.000, E1   +13.489, E3 +167982.784}
SPL {X  -160.000, Y  +631.625, Z    +0.000, E1   +13.508, E3 +168002.325}
SPL {X  -160.000, Y  +629.417, Z    +0.000, E1   +13.491, E3 +168021.936}
SPL {X  -160.000, Y  +627.180, Z    +0.000, E1   +13.508, E3 +168041.690}
SPL {X  -160.000, Y  +624.970, Z    +0.000, E1   +13.490, E3 +168061.340}
SPL {X  -160.000, Y  +623.020, Z    +0.000, E1   +13.491, E3 +168078.570}
SPL {X  -160.000, Y  +620.888, Z    +0.000, E1   +13.501, E3 +168097.432}
SPL {X  -160.000, Y  +618.790, Z    +0.000, E1   +13.488, E3 +168116.055}
SPL {X  -160.000, Y  +616.631, Z    +0.000, E1   +13.504, E3 +168135.108}
SPL {X  -160.000, Y  +614.230, Z    +0.000, E1   +13.510, E3 +168156.304}
SPL {X  -160.000, Y  +612.132, Z    +0.000, E1   +13.485, E3 +168175.021}
SPL {X  -160.000, Y  +610.405, Z    +0.000, E1   +13.477, E3 +168190.394}
SPL {X  -160.000, Y  +608.437, Z    +0.000, E1   +13.502, E3 +168207.649}
SPL {X  -160.000, Y  +606.281, Z    +0.000, E1   +13.502, E3 +168226.667}
SPL {X  -160.000, Y  +604.124, Z    +0.000, E1   +13.513, E3 +168245.722}
SPL {X  -160.000, Y  +601.878, Z    +0.000, E1   +13.505, E3 +168265.619}
SPL {X  -160.000, Y  +599.648, Z    +0.000, E1   +13.506, E3 +168285.396}
SPL {X  -160.000, Y  +597.673, Z    +0.000, E1   +13.479, E3 +168303.070}
SPL {X  -160.000, Y  +595.601, Z    +0.000, E1   +13.499, E3 +168321.353}
SPL {X  -160.000, Y  +593.187, Z    +0.000, E1   +13.500, E3 +168342.733}
SPL {X  -160.000, Y  +591.079, Z    +0.000, E1   +13.483, E3 +168361.459}
SPL {X  -160.000, Y  +589.151, Z    +0.000, E1   +13.489, E3 +168378.510}
SPL {X  -160.000, Y  +586.908, Z    +0.000, E1   +13.501, E3 +168398.356}
SPL {X  -160.000, Y  +584.660, Z    +0.000, E1   +13.490, E3 +168418.297}
SPL {X  -160.000, Y  +582.409, Z    +0.000, E1   +13.499, E3 +168438.215}
SPL {X  -160.000, Y  +580.150, Z    +0.000, E1   +13.490, E3 +168458.262}
SPL {X  -160.000, Y  +577.953, Z    +0.000, E1   +13.493, E3 +168477.720}
SPL {X  -160.000, Y  +575.630, Z    +0.000, E1   +13.502, E3 +168498.204}
SPL {X  -160.000, Y  +573.418, Z    +0.000, E1   +13.502, E3 +168517.712}
SPL {X  -160.000, Y  +571.226, Z    +0.000, E1   +13.520, E3 +168536.921}
SPL {X  -160.000, Y  +569.166, Z    +0.000, E1   +13.512, E3 +168555.111}
SPL {X  -160.000, Y  +567.275, Z    +0.000, E1   +13.517, E3 +168571.779}
SPL {X  -160.000, Y  +565.259, Z    +0.000, E1   +13.523, E3 +168589.568}
SPL {X  -160.000, Y  +563.305, Z    +0.000, E1   +13.512, E3 +168606.906}
SPL {X  -160.000, Y  +561.240, Z    +0.000, E1   +13.521, E3 +168625.168}
SPL {X  -160.000, Y  +558.881, Z    +0.000, E1   +13.524, E3 +168646.010}
SPL {X  -160.000, Y  +556.697, Z    +0.000, E1   +13.510, E3 +168665.396}
SPL {X  -160.000, Y  +554.624, Z    +0.000, E1   +13.512, E3 +168683.727}
SPL {X  -160.000, Y  +552.465, Z    +0.000, E1   +13.514, E3 +168702.811}
SPL {X  -160.000, Y  +550.315, Z    +0.000, E1   +13.514, E3 +168721.805}
SPL {X  -160.000, Y  +548.056, Z    +0.000, E1   +13.519, E3 +168741.806}
SPL {X  -160.000, Y  +545.826, Z    +0.000, E1   +13.501, E3 +168761.684}
SPL {X  -160.000, Y  +543.677, Z    +0.000, E1   +13.502, E3 +168780.741}
SPL {X  -160.000, Y  +541.664, Z    +0.000, E1   +13.489, E3 +168798.627}
SPL {X  -160.000, Y  +539.659, Z    +0.000, E1   +13.494, E3 +168816.387}
SPL {X  -160.000, Y  +537.370, Z    +0.000, E1   +13.501, E3 +168836.626}
SPL {X  -160.000, Y  +535.056, Z    +0.000, E1   +13.506, E3 +168857.022}
SPL {X  -160.000, Y  +532.975, Z    +0.000, E1   +13.494, E3 +168875.508}
SPL {X  -160.000, Y  +530.925, Z    +0.000, E1   +13.499, E3 +168893.670}
SPL {X  -160.000, Y  +528.768, Z    +0.000, E1   +13.498, E3 +168912.771}
SPL {X  -160.000, Y  +526.547, Z    +0.000, E1   +13.499, E3 +168932.440}
SPL {X  -160.000, Y  +523.964, Z    +0.000, E1   +13.742, E3 +168951.945}
SPL {X  -160.000, Y  +513.971, Z    +0.000, E1   +18.644, E3 +168970.857}
SPL {X  -160.000, Y  +513.562, Z    +0.000, E1   +16.972, E3 +168990.733}
SPL {X  -160.000, Y  +513.358, Z    +0.000, E1   +15.267, E3 +169011.005}
SPL {X  -160.000, Y  +512.244, Z    +0.000, E1   +14.473, E3 +169029.462}
SPL {X  -160.000, Y  +509.675, Z    +0.000, E1   +14.481, E3 +169050.605}
SPL {X  -160.000, Y  +507.162, Z    +0.000, E1   +14.470, E3 +169071.345}
SPL {X  -160.000, Y  +504.735, Z    +0.000, E1   +14.473, E3 +169091.316}
SPL {X  -160.000, Y  +502.261, Z    +0.000, E1   +14.476, E3 +169111.652}
SPL {X  -160.000, Y  +499.798, Z    +0.000, E1   +14.482, E3 +169131.855}
SPL {X  -160.000, Y  +497.435, Z    +0.000, E1   +14.476, E3 +169151.331}
SPL {X  -160.000, Y  +495.089, Z    +0.000, E1   +14.475, E3 +169170.698}
SPL {X  -160.000, Y  +492.764, Z    +0.000, E1   +14.469, E3 +169189.870}
SPL {X  -160.000, Y  +490.292, Z    +0.000, E1   +14.476, E3 +169210.271}
SPL {X  -160.000, Y  +487.641, Z    +0.000, E1   +14.470, E3 +169232.167}
SPL {X  -160.000, Y  +485.054, Z    +0.000, E1   +14.460, E3 +169253.609}
SPL {X  -160.000, Y  +482.421, Z    +0.000, E1   +14.461, E3 +169275.328}
SPL {X  -160.000, Y  +480.000, Z    +0.000, E1   +14.451, E3 +169295.292}
SPL {X  -160.000, Y  +477.551, Z    +0.000, E1   +14.466, E3 +169315.420}
SPL {X  -160.000, Y  +475.253, Z    +0.000, E1   +14.450, E3 +169334.395}
SPL {X  -160.000, Y  +473.070, Z    +0.000, E1   +14.454, E3 +169352.416}
SPL {X  -160.000, Y  +470.603, Z    +0.000, E1   +14.464, E3 +169372.716}
SPL {X  -160.000, Y  +468.243, Z    +0.000, E1   +14.458, E3 +169392.115}
SPL {X  -160.000, Y  +465.791, Z    +0.000, E1   +14.475, E3 +169412.259}
SPL {X  -160.000, Y  +463.103, Z    +0.000, E1   +14.474, E3 +169434.408}
SPL {X  -160.000, Y  +460.743, Z    +0.000, E1   +14.465, E3 +169453.816}
SPL {X  -160.000, Y  +458.292, Z    +0.000, E1   +14.492, E3 +169473.815}
SPL {X  -160.000, Y  +455.874, Z    +0.000, E1   +14.484, E3 +169493.673}
SPL {X  -160.000, Y  +453.555, Z    +0.000, E1   +14.488, E3 +169512.752}
SPL {X  -160.000, Y  +451.093, Z    +0.000, E1   +14.485, E3 +169533.064}
SPL {X  -160.000, Y  +448.700, Z    +0.000, E1   +14.483, E3 +169552.754}
SPL {X  -160.000, Y  +446.277, Z    +0.000, E1   +14.485, E3 +169572.677}
SPL {X  -160.000, Y  +443.879, Z    +0.000, E1   +14.485, E3 +169592.416}
SPL {X  -160.000, Y  +441.447, Z    +0.000, E1   +14.485, E3 +169612.423}
SPL {X  -160.000, Y  +439.006, Z    +0.000, E1   +14.488, E3 +169632.506}
SPL {X  -160.000, Y  +436.311, Z    +0.000, E1   +14.498, E3 +169654.665}
SPL {X  -160.000, Y  +433.559, Z    +0.000, E1   +14.491, E3 +169677.334}
SPL {X  -160.000, Y  +431.162, Z    +0.000, E1   +14.479, E3 +169697.085}
SPL {X  -160.000, Y  +429.152, Z    +0.000, E1   +14.469, E3 +169713.667}
SPL {X  -160.000, Y  +426.863, Z    +0.000, E1   +14.490, E3 +169732.446}
SPL {X  -160.000, Y  +424.653, Z    +0.000, E1   +14.467, E3 +169750.705}
SPL {X  -160.000, Y  +422.337, Z    +0.000, E1   +14.492, E3 +169769.689}
SPL {X  -160.000, Y  +419.639, Z    +0.000, E1   +14.504, E3 +169791.729}
SPL {X  -160.000, Y  +417.127, Z    +0.000, E1   +14.501, E3 +169812.321}
SPL {X  -160.000, Y  +414.849, Z    +0.000, E1   +14.496, E3 +169831.055}
SPL {X  -160.000, Y  +412.396, Z    +0.000, E1   +14.505, E3 +169851.243}
SPL {X  -160.000, Y  +409.815, Z    +0.000, E1   +14.498, E3 +169872.498}
SPL {X  -160.000, Y  +407.614, Z    +0.000, E1   +14.484, E3 +169890.623}
SPL {X  -160.000, Y  +405.406, Z    +0.000, E1   +14.501, E3 +169908.686}
SPL {X  -160.000, Y  +402.958, Z    +0.000, E1   +14.500, E3 +169928.856}
SPL {X  -160.000, Y  +400.690, Z    +0.000, E1   +14.484, E3 +169947.568}
SPL {X  -160.000, Y  +398.391, Z    +0.000, E1   +14.502, E3 +169966.394}
SPL {X  -160.000, Y  +395.999, Z    +0.000, E1   +14.484, E3 +169986.184}
SPL {X  -160.000, Y  +393.685, Z    +0.000, E1   +14.486, E3 +170005.256}
SPL {X  -159.999, Y  +391.313, Z    +0.000, E1   +14.479, E3 +170024.838}
SPL {X  -159.970, Y  +388.900, Z    +0.000, E1   +14.480, E3 +170044.722}
SPL {X  -159.903, Y  +386.417, Z    +0.000, E1   +14.475, E3 +170065.227}
SPL {X  -159.796, Y  +383.921, Z    +0.000, E1   +14.466, E3 +170085.883}
SPL {X  -159.651, Y  +381.443, Z    +0.000, E1   +14.453, E3 +170106.430}
SPL {X  -159.474, Y  +379.042, Z    +0.000, E1   +14.434, E3 +170126.395}
SPL {X  -159.316, Y  +377.219, Z    +0.000, E1   +14.400, E3 +170141.623}
ENDSPLINE

SPLINE
SPL {X  -159.452, Y  +378.767, Z    +0.000, E1   +11.887, E3 +170162.612}
SPL {X  -159.840, Y  +384.856, Z    +0.000, E1    +7.126, E3 +170181.584}
SPL {X  -159.991, Y  +390.336, Z    +0.000, E1    +2.803, E3 +170195.407}
SPL {X  -160.000, Y  +403.532, Z    +0.000, E1    -6.523, E3 +170213.127}
SPL {X  -160.000, Y  +409.023, Z    +0.000, E1   -10.003, E3 +170223.901}
SPL {X  -160.000, Y  +418.032, Z    +0.000, E1   -14.569, E3 +170248.760}
SPL {X  -160.000, Y  +420.561, Z    +0.000, E1   -14.816, E3 +170266.240}
SPL {X  -160.000, Y  +422.801, Z    +0.000, E1   -14.823, E3 +170284.189}
SPL {X  -160.000, Y  +425.518, Z    +0.000, E1   -14.845, E3 +170305.963}
SPL {X  -160.000, Y  +428.688, Z    +0.000, E1   -14.854, E3 +170331.371}
SPL {X  -160.000, Y  +431.971, Z    +0.000, E1   -14.849, E3 +170357.840}
SPL {X  -160.000, Y  +435.345, Z    +0.000, E1   -14.857, E3 +170384.890}
SPL {X  -160.000, Y  +438.732, Z    +0.000, E1   -14.858, E3 +170412.039}
SPL {X  -160.000, Y  +441.925, Z    +0.000, E1   -14.848, E3 +170437.709}
SPL {X  -160.000, Y  +444.299, Z    +0.000, E1   -14.809, E3 +170456.894}
SPL {X  -160.000, Y  +446.229, Z    +0.000, E1   -14.820, E3 +170472.313}
SPL {X  -160.000, Y  +448.987, Z    +0.000, E1   -14.868, E3 +170494.249}
SPL {X  -160.000, Y  +452.351, Z    +0.000, E1   -14.871, E3 +170521.225}
SPL {X  -160.000, Y  +455.709, Z    +0.000, E1   -14.880, E3 +170548.039}
SPL {X  -160.000, Y  +458.189, Z    +0.000, E1   -14.832, E3 +170568.041}
SPL {X  -160.000, Y  +459.885, Z    +0.000, E1   -14.825, E3 +170581.712}
SPL {X  -160.000, Y  +462.438, Z    +0.000, E1   -14.868, E3 +170602.122}
SPL {X  -160.000, Y  +465.575, Z    +0.000, E1   -14.849, E3 +170627.430}
SPL {X  -160.000, Y  +468.581, Z    +0.000, E1   -14.841, E3 +170651.662}
SPL {X  -160.000, Y  +471.795, Z    +0.000, E1   -14.854, E3 +170677.450}
SPL {X  -160.000, Y  +475.138, Z    +0.000, E1   -14.853, E3 +170704.300}
SPL {X  -160.000, Y  +477.981, Z    +0.000, E1   -14.823, E3 +170727.220}
SPL {X  -160.000, Y  +480.658, Z    +0.000, E1   -14.835, E3 +170748.696}
SPL {X  -160.000, Y  +483.534, Z    +0.000, E1   -14.838, E3 +170771.791}
SPL {X  -160.000, Y  +486.226, Z    +0.000, E1   -14.823, E3 +170793.456}
SPL {X  -160.000, Y  +488.751, Z    +0.000, E1   -14.827, E3 +170813.729}
SPL {X  -160.000, Y  +491.612, Z    +0.000, E1   -14.844, E3 +170836.651}
SPL {X  -160.000, Y  +494.417, Z    +0.000, E1   -14.827, E3 +170859.242}
SPL {X  -160.000, Y  +496.961, Z    +0.000, E1   -14.824, E3 +170879.686}
SPL {X  -160.000, Y  +499.610, Z    +0.000, E1   -14.830, E3 +170900.959}
SPL {X  -160.000, Y  +502.268, Z    +0.000, E1   -14.832, E3 +170922.228}
SPL {X  -160.000, Y  +505.041, Z    +0.000, E1   -14.849, E3 +170944.390}
SPL {X  -160.000, Y  +507.743, Z    +0.000, E1   -14.842, E3 +170966.014}
SPL {X  -160.000, Y  +510.437, Z    +0.000, E1   -14.860, E3 +170987.528}
SPL {X  -160.000, Y  +513.179, Z    +0.000, E1   -14.849, E3 +171009.576}
SPL {X  -160.000, Y  +515.613, Z    +0.000, E1   -14.829, E3 +171029.246}
SPL {X  -160.000, Y  +518.188, Z    +0.000, E1   -14.845, E3 +171049.875}
SPL {X  -160.000, Y  +520.790, Z    +0.000, E1   -14.839, E3 +171070.704}
SPL {X  -160.000, Y  +523.469, Z    +0.000, E1   -14.855, E3 +171092.152}
SPL {X  -160.000, Y  +526.403, Z    +0.000, E1   -14.858, E3 +171115.689}
SPL {X  -160.000, Y  +529.266, Z    +0.000, E1   -14.848, E3 +171138.696}
SPL {X  -160.000, Y  +531.688, Z    +0.000, E1   -14.826, E3 +171158.246}
SPL {X  -160.000, Y  +534.214, Z    +0.000, E1   -14.841, E3 +171178.509}
SPL {X  -160.000, Y  +537.002, Z    +0.000, E1   -14.839, E3 +171200.927}
SPL {X  -160.000, Y  +539.729, Z    +0.000, E1   -14.840, E3 +171222.739}
SPL {X  -160.000, Y  +542.408, Z    +0.000, E1   -14.839, E3 +171244.292}
SPL {X  -160.000, Y  +545.014, Z    +0.000, E1   -14.831, E3 +171265.237}
SPL {X  -160.000, Y  +547.659, Z    +0.000, E1   -14.839, E3 +171286.451}
SPL {X  -160.000, Y  +550.215, Z    +0.000, E1   -14.827, E3 +171307.016}
SPL {X  -160.000, Y  +552.762, Z    +0.000, E1   -14.836, E3 +171327.435}
SPL {X  -160.000, Y  +555.331, Z    +0.000, E1   -14.837, E3 +171347.976}
SPL {X  -160.000, Y  +558.235, Z    +0.000, E1   -14.869, E3 +171371.139}
SPL {X  -160.000, Y  +561.088, Z    +0.000, E1   -14.848, E3 +171394.058}
SPL {X  -160.000, Y  +563.693, Z    +0.000, E1   -14.852, E3 +171414.918}
SPL {X  -160.000, Y  +566.560, Z    +0.000, E1   -14.865, E3 +171437.896}
SPL {X  -160.000, Y  +569.305, Z    +0.000, E1   -14.848, E3 +171459.924}
SPL {X  -160.000, Y  +571.769, Z    +0.000, E1   -14.852, E3 +171479.670}
SPL {X  -160.000, Y  +574.366, Z    +0.000, E1   -14.855, E3 +171500.457}
SPL {X  -160.000, Y  +577.037, Z    +0.000, E1   -14.859, E3 +171521.857}
SPL {X  -160.000, Y  +579.855, Z    +0.000, E1   -14.869, E3 +171544.384}
SPL {X  -160.000, Y  +582.456, Z    +0.000, E1   -14.854, E3 +171565.244}
SPL {X  -160.000, Y  +585.083, Z    +0.000, E1   -14.866, E3 +171586.293}
SPL {X  -160.000, Y  +587.675, Z    +0.000, E1   -14.853, E3 +171607.084}
SPL {X  -160.000, Y  +590.216, Z    +0.000, E1   -14.864, E3 +171627.404}
SPL {X  -160.000, Y  +592.848, Z    +0.000, E1   -14.865, E3 +171648.455}
SPL {X  -160.000, Y  +595.342, Z    +0.000, E1   -14.848, E3 +171668.632}
SPL {X  -160.000, Y  +597.995, Z    +0.000, E1   -14.848, E3 +171689.972}
SPL {X  -160.000, Y  +600.731, Z    +0.000, E1   -14.846, E3 +171711.924}
SPL {X  -160.000, Y  +603.404, Z    +0.000, E1   -14.846, E3 +171733.359}
SPL {X  -160.000, Y  +605.923, Z    +0.000, E1   -14.838, E3 +171753.600}
SPL {X  -160.000, Y  +608.492, Z    +0.000, E1   -14.846, E3 +171774.204}
SPL {X  -160.000, Y  +611.345, Z    +0.000, E1   -14.856, E3 +171797.062}
SPL {X  -160.000, Y  +614.087, Z    +0.000, E1   -14.839, E3 +171819.122}
SPL {X  -160.000, Y  +616.566, Z    +0.000, E1   -14.839, E3 +171839.015}
SPL {X  -160.000, Y  +619.350, Z    +0.000, E1   -14.855, E3 +171861.303}
SPL {X  -160.000, Y  +622.198, Z    +0.000, E1   -14.846, E3 +171884.188}
SPL {X  -160.000, Y  +624.642, Z    +0.000, E1   -14.829, E3 +171903.861}
SPL {X  -160.000, Y  +627.119, Z    +0.000, E1   -14.843, E3 +171923.700}
SPL {X  -160.000, Y  +629.682, Z    +0.000, E1   -14.838, E3 +171944.269}
SPL {X  -160.000, Y  +632.223, Z    +0.000, E1   -14.841, E3 +171964.661}
SPL {X  -160.000, Y  +634.941, Z    +0.000, E1   -14.846, E3 +171986.458}
SPL {X  -160.000, Y  +637.723, Z    +0.000, E1   -14.844, E3 +172008.802}
SPL {X  -160.000, Y  +640.315, Z    +0.000, E1   -14.836, E3 +172029.600}
SPL {X  -160.000, Y  +643.085, Z    +0.000, E1   -14.865, E3 +172051.652}
SPL {X  -160.000, Y  +645.845, Z    +0.000, E1   -14.848, E3 +172073.840}
SPL {X  -160.000, Y  +648.229, Z    +0.000, E1   -14.834, E3 +172093.049}
SPL {X  -160.000, Y  +650.656, Z    +0.000, E1   -14.835, E3 +172112.606}
SPL {X  -160.000, Y  +653.134, Z    +0.000, E1   -14.827, E3 +172132.533}
SPL {X  -160.000, Y  +655.670, Z    +0.000, E1   -14.841, E3 +172152.827}
SPL {X  -160.000, Y  +658.349, Z    +0.000, E1   -14.842, E3 +172174.302}
SPL {X  -160.000, Y  +660.936, Z    +0.000, E1   -14.838, E3 +172195.054}
SPL {X  -160.000, Y  +663.567, Z    +0.000, E1   -14.845, E3 +172216.185}
SPL {X  -160.000, Y  +666.216, Z    +0.000, E1   -14.832, E3 +172237.501}
SPL {X  -159.997, Y  +668.731, Z    +0.000, E1   -14.834, E3 +172257.693}
SPL {X  -159.962, Y  +671.176, Z    +0.000, E1   -14.822, E3 +172277.404}
SPL {X  -159.895, Y  +673.507, Z    +0.000, E1   -14.821, E3 +172296.136}
SPL {X  -159.785, Y  +675.985, Z    +0.000, E1   -14.818, E3 +172316.137}
SPL {X  -159.627, Y  +678.622, Z    +0.000, E1   -14.804, E3 +172337.490}
SPL {X  -159.438, Y  +681.094, Z    +0.000, E1   -14.770, E3 +172357.661}
SPL {X  -159.262, Y  +683.054, Z    +0.000, E1   -14.719, E3 +172373.890}
ENDSPLINE

SPLINE
SPL {X  -159.661, Y  +678.114, Z    +0.000, E1    -9.575, E3 +172403.482}
SPL {X  -159.942, Y  +672.020, Z    +0.000, E1    -4.692, E3 +172422.109}
SPL {X  -160.000, Y  +664.971, Z    +0.000, E1    +0.516, E3 +172441.659}
SPL {X  -160.000, Y  +660.032, Z    +0.000, E1    +3.995, E3 +172453.602}
SPL {X  -160.000, Y  +652.280, Z    +0.000, E1    +8.913, E3 +172472.117}
SPL {X  -160.000, Y  +644.147, Z    +0.000, E1   +13.158, E3 +172495.667}
SPL {X  -160.000, Y  +641.594, Z    +0.000, E1   +13.488, E3 +172514.108}
SPL {X  -160.000, Y  +639.799, Z    +0.000, E1   +13.486, E3 +172530.018}
SPL {X  -160.000, Y  +637.896, Z    +0.000, E1   +13.493, E3 +172546.833}
SPL {X  -160.000, Y  +635.832, Z    +0.000, E1   +13.499, E3 +172565.092}
SPL {X  -160.000, Y  +633.839, Z    +0.000, E1   +13.489, E3 +172582.781}
SPL {X  -160.000, Y  +631.625, Z    +0.000, E1   +13.508, E3 +172602.322}
SPL {X  -160.000, Y  +629.417, Z    +0.000, E1   +13.491, E3 +172621.933}
SPL {X  -160.000, Y  +627.180, Z    +0.000, E1   +13.508, E3 +172641.687}
SPL {X  -160.000, Y  +624.970, Z    +0.000, E1   +13.490, E3 +172661.337}
SPL {X  -160.000, Y  +623.020, Z    +0.000, E1   +13.491, E3 +172678.567}
SPL {X  -160.000, Y  +620.888, Z    +0.000, E1   +13.501, E3 +172697.429}
SPL {X  -160.000, Y  +618.790, Z    +0.000, E1   +13.488, E3 +172716.052}
SPL {X  -160.000, Y  +616.631, Z    +0.000, E1   +13.504, E3 +172735.105}
SPL {X  -160.000, Y  +614.230, Z    +0.000, E1   +13.510, E3 +172756.301}
SPL {X  -160.000, Y  +612.132, Z    +0.000, E1   +13.485, E3 +172775.017}
SPL {X  -160.000, Y  +610.405, Z    +0.000, E1   +13.477, E3 +172790.391}
SPL {X  -160.000, Y  +608.437, Z    +0.000, E1   +13.502, E3 +172807.646}
SPL {X  -160.000, Y  +606.281, Z    +0.000, E1   +13.502, E3 +172826.664}
SPL {X  -160.000, Y  +604.124, Z    +0.000, E1   +13.513, E3 +172845.719}
SPL {X  -160.000, Y  +601.878, Z    +0.000, E1   +13.505, E3 +172865.616}
SPL {X  -160.000, Y  +599.648, Z    +0.000, E1   +13.506, E3 +172885.393}
SPL {X  -160.000, Y  +597.673, Z    +0.000, E1   +13.479, E3 +172903.066}
SPL {X  -160.000, Y  +595.601, Z    +0.000, E1   +13.499, E3 +172921.350}
SPL {X  -160.000, Y  +593.187, Z    +0.000, E1   +13.500, E3 +172942.730}
SPL {X  -160.000, Y  +591.079, Z    +0.000, E1   +13.483, E3 +172961.456}
SPL {X  -160.000, Y  +589.151, Z    +0.000, E1   +13.489, E3 +172978.507}
SPL {X  -160.000, Y  +586.908, Z    +0.000, E1   +13.501, E3 +172998.352}
SPL {X  -160.000, Y  +584.660, Z    +0.000, E1   +13.490, E3 +173018.294}
SPL {X  -160.000, Y  +582.409, Z    +0.000, E1   +13.499, E3 +173038.212}
SPL {X  -160.000, Y  +580.150, Z    +0.000, E1   +13.490, E3 +173058.259}
SPL {X  -160.000, Y  +577.953, Z    +0.000, E1   +13.493, E3 +173077.717}
SPL {X  -160.000, Y  +575.630, Z    +0.000, E1   +13.502, E3 +173098.201}
SPL {X  -160.000, Y  +573.418, Z    +0.000, E1   +13.502, E3 +173117.709}
SPL {X  -160.000, Y  +571.226, Z    +0.000, E1   +13.520, E3 +173136.918}
SPL {X  -160.000, Y  +569.166, Z    +0.000, E1   +13.512, E3 +173155.108}
SPL {X  -160.000, Y  +567.275, Z    +0.000, E1   +13.517, E3 +173171.775}
SPL {X  -160.000, Y  +565.259, Z    +0.000, E1   +13.523, E3 +173189.565}
SPL {X  -160.000, Y  +563.305, Z    +0.000, E1   +13.512, E3 +173206.903}
SPL {X  -160.000, Y  +561.240, Z    +0.000, E1   +13.521, E3 +173225.164}
SPL {X  -160.000, Y  +558.881, Z    +0.000, E1   +13.524, E3 +173246.007}
SPL {X  -160.000, Y  +556.697, Z    +0.000, E1   +13.510, E3 +173265.393}
SPL {X  -160.000, Y  +554.624, Z    +0.000, E1   +13.512, E3 +173283.724}
SPL {X  -160.000, Y  +552.465, Z    +0.000, E1   +13.514, E3 +173302.808}
SPL {X  -160.000, Y  +550.315, Z    +0.000, E1   +13.514, E3 +173321.802}
SPL {X  -160.000, Y  +548.056, Z    +0.000, E1   +13.519, E3 +173341.803}
SPL {X  -160.000, Y  +545.826, Z    +0.000, E1   +13.501, E3 +173361.680}
SPL {X  -160.000, Y  +543.677, Z    +0.000, E1   +13.502, E3 +173380.738}
SPL {X  -160.000, Y  +541.664, Z    +0.000, E1   +13.489, E3 +173398.624}
SPL {X  -160.000, Y  +539.659, Z    +0.000, E1   +13.494, E3 +173416.384}
SPL {X  -160.000, Y  +537.370, Z    +0.000, E1   +13.501, E3 +173436.623}
SPL {X  -160.000, Y  +535.056, Z    +0.000, E1   +13.506, E3 +173457.018}
SPL {X  -160.000, Y  +532.975, Z    +0.000, E1   +13.494, E3 +173475.505}
SPL {X  -160.000, Y  +530.925, Z    +0.000, E1   +13.499, E3 +173493.667}
SPL {X  -160.000, Y  +528.768, Z    +0.000, E1   +13.498, E3 +173512.768}
SPL {X  -160.000, Y  +526.547, Z    +0.000, E1   +13.499, E3 +173532.437}
SPL {X  -160.000, Y  +523.964, Z    +0.000, E1   +13.742, E3 +173551.941}
SPL {X  -160.000, Y  +513.971, Z    +0.000, E1   +18.644, E3 +173570.853}
SPL {X  -160.000, Y  +513.562, Z    +0.000, E1   +16.972, E3 +173590.730}
SPL {X  -160.000, Y  +513.358, Z    +0.000, E1   +15.267, E3 +173611.006}
ENDSPLINE
END
